FUNCTION proj1_TupleStruct_1: DINT
{ S7_Optimized_Access := 'false' }
    VAR_INPUT
        tuple: TupleStruct_1;
    END_VAR

BEGIN
    proj1_TupleStruct_1 := tuple.field1;
END_FUNCTION
